FUNCTION_BLOCK PUBLIC FB_SubjectNew EXTENDS FB_Base IMPLEMENTS I_Subject
VAR
	fbDelay				: TON;
	fbDrand				: DRAND;
	fValue				: LREAL;
	fbSubjectBase		: FB_SubjectBase;
END_VAR

// creates every sec a random value and invoke the update method
fbDelay(IN := TRUE, PT := T#500MS);
IF (fbDelay.Q) THEN	
	fbDelay(IN := FALSE);
	fbDrand(SEED := TO_INT(ADR(fValue)));
	fValue := fbDrand.Num * 1.0;
	THIS^.Notify();
END_IF

METHOD PUBLIC Attach : BOOL
VAR_INPUT
	ipObserver				: I_Observer;
END_VAR
Attach := FALSE;
IF (THIS^.fbSubjectBase.Attach(ipObserver)) THEN
	ipObserver.Update(THIS^.fValue);
	Attach := TRUE;
END_IF
END_METHOD

METHOD PUBLIC Detach : BOOL
VAR_INPUT
	ipObserver		: I_Observer;
END_VAR
Detach := THIS^.fbSubjectBase.Detach(ipObserver);
END_METHOD

{attribute 'monitoring':='call'}
PROPERTY PUBLIC fActualValue : LREAL
GET
fActualValue := THIS^.fValue;
END_GET
END_PROPERTY

METHOD PRIVATE Notify
VAR	
	nIndex		: INT := 0;
END_VAR
FOR nIndex := 1 TO Param.cMaxObservers DO
	IF (THIS^.fbSubjectBase.aObservers[nIndex] <> 0) THEN
		THIS^.fbSubjectBase.aObservers[nIndex].Update(THIS^.fActualValue);
	END_IF
END_FOR
END_METHOD

END_FUNCTION_BLOCK

(* stored: Version 1.1.0.1, ProductVersion 3.1.4022.10
   POU FB_SubjectNew: Id {02cbaef6-009b-4e16-a3e9-0a9408536e35}, SpecialFunc None
   Method Attach: Id {e41e34e6-7327-467e-aa5c-96bda1aafde4}
   Method Detach: Id {8e131d16-7352-4f70-badb-52803a6e195e}
   Property fActualValue: Id {eff8a6a5-e699-4aa2-ab1d-31af949b37ae}
   Get Get: Id {9c23695c-45ab-4175-83e8-5fd7d75c008f}
   Method Notify: Id {73845a56-27bf-4b99-8966-8d5dd109eb49} *)
